Yaskawa INFORM job: trapez_05_05_2024_planes_program.JBI

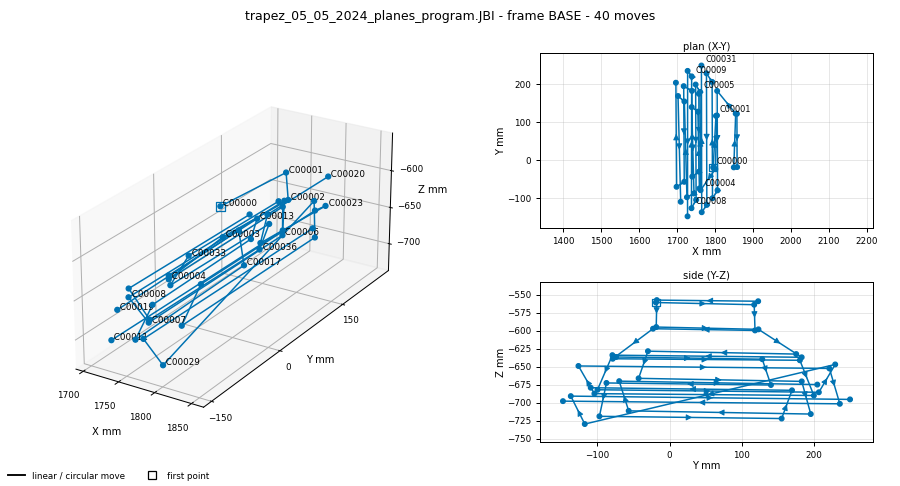
[picture p0: tool path of trapez_05_05_2024_planes_program.JBI in frame BASE, 40 of 45 moves have a stored position in this frame; points joined in program order, loops and branches not executed]
/JOB
//NAME trapez_05_05_2024_planes_program
//POS
///NPOS 40,0,40,0,0,0
///TOOL 0
///POSTYPE BASE
///RECTAN
///RCONF 0,0,0,0,0,0,0,0,0,0,0,0,0,0,0,0,0,0,0,0,0,0,0,0
C00000=1795.615174,-18.972207,-560.999386,175.000000,-76.567719,-5.000000
C00001=1802.947639,117.188673,-564.042088,175.000000,-76.567719,-5.000000
C00002=1805.566371,118.303086,-599.679746,175.000000,-76.567719,-5.000000
C00003=1801.208361,-23.007539,-597.298583,175.000000,-76.567719,-5.000000
C00004=1762.458100,-78.842155,-638.922692,175.000000,-76.567719,-5.000000
C00005=1760.972186,180.445841,-641.027182,175.000000,-76.567719,-5.000000
C00006=1749.318372,199.863012,-689.836483,175.000000,-76.567719,-5.000000
C00007=1750.623670,-104.253462,-687.263654,175.000000,-76.567719,-5.000000
C00008=1738.357975,-126.347153,-648.930545,175.000000,-76.567719,-5.000000
C00009=1738.830774,221.381887,-652.341704,175.000000,-76.567719,-5.000000
C00010=1728.229006,235.848401,-701.355307,175.000000,-76.567719,-5.000000
C00011=1727.996544,-147.802391,-697.660826,180.000000,-60.000000,0.000000
C00012=1759.260461,-74.232505,-636.474689,175.000000,-68.536690,-5.000000
C00013=1755.291086,128.357064,-639.528973,175.000000,-68.536690,-5.000000
C00014=1739.000904,140.367800,-675.296665,175.000000,-68.536690,-5.000000
C00015=1744.991793,-87.534673,-672.460584,175.000000,-68.536690,-5.000000
C00016=1726.421778,-97.293960,-718.674923,175.000000,-68.536690,-5.000000
C00017=1719.627571,155.222685,-721.755864,175.000000,-68.536690,-5.000000
C00018=1702.896300,169.564378,-682.639613,175.000000,-68.536690,-5.000000
C00019=1709.917189,-109.336141,-679.046784,180.000000,-60.000000,0.000000
C00020=1858.202243,122.701683,-559.228409,175.000000,-73.932600,-5.000000
C00021=1858.705443,-17.761817,-557.639860,175.000000,-73.932600,-5.000000
C00022=1849.955146,-18.579481,-594.982159,175.000000,-73.932600,-5.000000
C00023=1854.964933,123.092668,-598.173467,175.000000,-73.932600,-5.000000
C00024=1806.097496,182.980220,-636.874018,175.000000,-73.932600,-5.000000
C00025=1807.120883,-79.312650,-633.931782,175.000000,-73.932600,-5.000000
C00026=1793.794883,-99.961927,-681.875024,175.000000,-73.932600,-5.000000
C00027=1792.780245,206.766429,-685.368165,175.000000,-73.932600,-5.000000
C00028=1777.910216,229.442945,-646.798847,175.000000,-73.932600,-5.000000
C00029=1778.866032,-117.574486,-729.394092,175.000000,-73.932600,-5.000000
C00030=1765.397324,-136.945204,-690.709471,175.000000,-73.932600,-5.000000
C00031=1764.591036,249.980287,-695.252343,180.000000,-60.000000,0.000000
C00032=1757.836251,175.402017,-632.443394,175.000000,-64.774545,-5.000000
C00033=1758.164526,-30.042628,-628.422990,175.000000,-64.774545,-5.000000
C00034=1740.431270,-42.990161,-666.051809,175.000000,-64.774545,-5.000000
C00035=1739.645908,183.063092,-670.275706,175.000000,-64.774545,-5.000000
C00036=1717.865584,195.573248,-715.549153,175.000000,-64.774545,-5.000000
C00037=1719.314035,-56.734343,-711.104098,175.000000,-64.774545,-5.000000
C00038=1699.019509,-69.851927,-669.954164,175.000000,-64.774545,-5.000000
C00039=1697.268336,204.651399,-674.707669,180.000000,-60.000000,0.000000
///POSTYPE PULSE
///PULSE
EC00000=4096.0
EC00001=4096.0
EC00002=4096.0
EC00003=4096.0
EC00004=4096.0
EC00005=4096.0
EC00006=4096.0
EC00007=4096.0
EC00008=4096.0
EC00009=4096.0
EC00010=4096.0
EC00011=4096.0
EC00012=98304.0
EC00013=98304.0
EC00014=98304.0
EC00015=98304.0
EC00016=98304.0
EC00017=98304.0
EC00018=98304.0
EC00019=98304.0
EC00020=189440.0
EC00021=189440.0
EC00022=189440.0
EC00023=189440.0
EC00024=189440.0
EC00025=189440.0
EC00026=189440.0
EC00027=189440.0
EC00028=189440.0
EC00029=189440.0
EC00030=189440.0
EC00031=189440.0
EC00032=281600.0
EC00033=281600.0
EC00034=281600.0
EC00035=281600.0
EC00036=281600.0
EC00037=281600.0
EC00038=281600.0
EC00039=281600.0
//INST
///DATE 2023/07/05 10:40
///ATTR SC,RW,RJ
////FRAME BASE
///GROUP1 RB1,ST1
NOP
MOVJ P009 EX000 VJ=15.00
MOVJ C00000 EC00000 VJ=15.0
CALL JOB:SPYON
MOVL C00001 EC00001 V=150.0
MOVL C00002 EC00002 V=150.0
MOVL C00003 EC00003 V=150.0
MOVL C00004 EC00004 V=150.0
MOVL C00005 EC00005 V=150.0
MOVL C00006 EC00006 V=150.0
MOVL C00007 EC00007 V=150.0
MOVL C00008 EC00008 V=150.0
MOVL C00009 EC00009 V=150.0
MOVL C00010 EC00010 V=150.0
MOVL C00011 EC00011 V=150.0
CALL JOB:SPYOF
MOVJ P009 VJ=15.00
MOVJ C00012 EC00012 VJ=15.0
CALL JOB:SPYON
MOVL C00013 EC00013 V=150.0
MOVL C00014 EC00014 V=150.0
MOVL C00015 EC00015 V=150.0
MOVL C00016 EC00016 V=150.0
MOVL C00017 EC00017 V=150.0
MOVL C00018 EC00018 V=150.0
MOVL C00019 EC00019 V=150.0
CALL JOB:SPYOF
MOVJ P009 VJ=15.00
MOVJ C00020 EC00020 VJ=15.0
CALL JOB:SPYON
MOVL C00021 EC00021 V=150.0
MOVL C00022 EC00022 V=150.0
MOVL C00023 EC00023 V=150.0
MOVL C00024 EC00024 V=150.0
MOVL C00025 EC00025 V=150.0
MOVL C00026 EC00026 V=150.0
MOVL C00027 EC00027 V=150.0
MOVL C00028 EC00028 V=150.0
MOVL C00029 EC00029 V=150.0
MOVL C00030 EC00030 V=150.0
MOVL C00031 EC00031 V=150.0
CALL JOB:SPYOF
MOVJ P009 VJ=15.00
MOVJ C00032 EC00032 VJ=15.0
CALL JOB:SPYON
MOVL C00033 EC00033 V=150.0
MOVL C00034 EC00034 V=150.0
MOVL C00035 EC00035 V=150.0
MOVL C00036 EC00036 V=150.0
MOVL C00037 EC00037 V=150.0
MOVL C00038 EC00038 V=150.0
MOVL C00039 EC00039 V=150.0
CALL JOB:SPYOF
MOVJ P009 VJ=15.00
END
